PROGRAM MAIN
VAR
	_defaultContext : DefaultContext;
END_VAR

_defaultContext.Run();

END_PROGRAM

(* stored: Version 1.1.0.1, ProductVersion 3.1.4024.6
   POU MAIN: Id {6d949533-a6b9-47e3-b85f-8c626bcf836e}, SpecialFunc None *)
